PROGRAM MAIN
VAR
	testConversion : UnitConversion_TestSuite;
END_VAR

TcUnit.RUN_IN_SEQUENCE();

END_PROGRAM

(* stored: Version 1.1.0.1
   POU MAIN: Id {e2000657-0558-4cd5-b540-68f1b2db8ff5}, SpecialFunc None *)
